// Mitsubishi GX Works2 project: BookEX6_18 Shift   PLC: Q13UDV

// global labels: Global
VAR_GLOBAL
  bVar0 AT M5000 : BOOL;
  abArray0 AT M5010 : ARRAY [0..49] OF BOOL;
  sStr0 AT D5000 : STRING[199];
  sStr1 AT D5100 : STRING[199];
  sStr2 AT D5200 : STRING[199];
  sStr3 AT D5300 : STRING[199];
  sStr4 AT D5400 : STRING[199];
  sStr5 AT D5500 : STRING[199];
  sStr6 AT D5600 : STRING[199];
  sStr7 AT D5700 : STRING[199];
  sStr8 AT D5800 : STRING[199];
  sStr9 AT D5900 : STRING[199];
  iVar0 AT D4500 : INT;
  iVar1 AT D4501 : INT;
  iVar2 AT D4502 : INT;
  iVar3 AT D4503 : INT;
  iVar4 AT D4504 : INT;
  iVar5 AT D4505 : INT;
  iVar6 AT D4506 : INT;
  iVar7 AT D4507 : INT;
  iVar8 AT D4508 : INT;
  iVar9 AT D4509 : INT;
  dVar0 AT D4510 : DINT;
  dVar1 AT D4512 : DINT;
  dVar2 AT D4514 : DINT;
  dVar3 AT D4516 : DINT;
  dVar4 AT D4518 : DINT;
  dVar5 AT D4520 : DINT;
  dVar6 AT D4522 : DINT;
  dVar7 AT D4524 : DINT;
  dVar8 AT D4526 : DINT;
  dVar9 AT D4528 : DINT;
  wVar0 AT D4530 : WORD;
  wVar1 AT D4531 : WORD;
  wVar2 AT D4532 : WORD;
  wVar3 AT D4533 : WORD;
  wVar4 AT D4534 : WORD;
  wVar5 AT D4535 : WORD;
  wVar6 AT D4536 : WORD;
  wVar7 AT D4537 : WORD;
  wVar8 AT D4538 : WORD;
  wVar9 AT D4539 : WORD;
  dwVar0 AT D4540 : DWORD;
  dwVar1 AT D4542 : DWORD;
  dwVar2 AT D4544 : DWORD;
  dwVar3 AT D4546 : DWORD;
  dwVar4 AT D4548 : DWORD;
  dwVar5 AT D4550 : DWORD;
  dwVar6 AT D4552 : DWORD;
  dwVar7 AT D4554 : DWORD;
  dwVar8 AT D4556 : DWORD;
  dwVar9 AT D4558 : DWORD;
  fsVar0 AT D4560 : REAL;
  fsVar1 AT D4562 : REAL;
  fsVar2 AT D4564 : REAL;
  fsVar3 AT D4566 : REAL;
  fsVar4 AT D4568 : REAL;
  fsVar5 AT D4570 : REAL;
  fsVar6 AT D4572 : REAL;
  fsVar7 AT D4574 : REAL;
  fsVar8 AT D4576 : REAL;
  fsVar9 AT D4578 : REAL;
  fdVar0 AT D4580 : LREAL;
  tTime0 AT D4620 : TIME;
  tTime1 AT D4622 : TIME;
  tTime2 AT D4624 : TIME;
  tTime3 AT D4626 : TIME;
  tTime4 AT D4628 : TIME;
  tTime5 AT D4630 : TIME;
  tTime6 AT D4632 : TIME;
  tTime7 AT D4634 : TIME;
  tTime8 AT D4636 : TIME;
  tTime9 AT D4638 : TIME;
  tTime10 AT D4640 : TIME;
  bVar1 AT M5001 : BOOL;
  bVar2 AT M5002 : BOOL;
  bVar3 AT M5003 : BOOL;
  bVar4 AT M5004 : BOOL;
  bVar5 AT M5005 : BOOL;
  bVar6 AT M5006 : BOOL;
  bVar7 AT M5007 : BOOL;
  bVar8 AT M5008 : BOOL;
  bVar9 AT M5009 : BOOL;
  abArray1 AT M5060 : ARRAY [0..49] OF BOOL;
  abArray2 AT M5110 : ARRAY [0..49] OF BOOL;
  abArray3 AT M5160 : ARRAY [0..49] OF BOOL;
  abArray4 AT M5210 : ARRAY [0..49] OF BOOL;
  abArray5 AT M5260 : ARRAY [0..49] OF BOOL;
  abArray6 AT M5310 : ARRAY [0..49] OF BOOL;
  abArray7 AT M5360 : ARRAY [0..49] OF BOOL;
  abArray8 AT M5410 : ARRAY [0..49] OF BOOL;
  abArray9 AT M5460 : ARRAY [0..49] OF BOOL;
  fdVar1 AT D4584 : LREAL;
  fdVar2 AT D4588 : LREAL;
  fdVar3 AT D4592 : LREAL;
  fdVar4 AT D4596 : LREAL;
  fdVar5 AT D4600 : LREAL;
  fdVar6 AT D4604 : LREAL;
  fdVar7 AT D4608 : LREAL;
  fdVar8 AT D4612 : LREAL;
  fdVar9 AT D4616 : LREAL;
  aSendData1 AT D100 : ARRAY [0..9] OF INT;
  aiTxData AT D4000 : ARRAY [0..99] OF INT;
  aiRxData AT D4100 : ARRAY [0..99] OF INT;
  iOpenOK AT D3900 : INT;
  iOpenERR AT D3901 : INT;
  iSendOK AT D3902 : INT;
  iSendERR AT D3903 : INT;
  iCloseOK AT D3906 : INT;
  iCloseERR AT D3907 : INT;
  iRecvOK AT D3904 : INT;
  iRecvERR AT D3905 : INT;
  aiTxData2 AT D4200 : ARRAY [0..99] OF INT;
  aiRxData2 AT D4300 : ARRAY [0..99] OF INT;
  iOpenOK2 AT D3908 : INT;
  iOpenERR2 AT D3909 : INT;
  iSendOK2 AT D3910 : INT;
  iSendERR2 AT D3911 : INT;
  iRecvOK2 AT D3912 : INT;
  iRecvERR2 AT D3913 : INT;
  iCloseOK2 AT D3914 : INT;
  iCloseERR2 AT D3915 : INT;
  iEOpenComp AT D3916 : INT;
  iEOpenReq AT D3917 : INT;
  iERecvFlag AT D3918 : INT;
  iOpenCode AT D3919 : INT;
  iSendCode AT D3920 : INT;
  iRecvCode AT D3921 : INT;
  iCloseCode AT D3922 : INT;
  iOpenCode2 AT D3923 : INT;
  iSendCode2 AT D3924 : INT;
  iRecvCode2 AT D3925 : INT;
  iCloseCode2 AT D3926 : INT;
  aRecvData1 AT D110 : ARRAY [0..9] OF INT;
  aSendData2 AT D120 : ARRAY [0..9] OF INT;
  aRecvData2 AT D130 : ARRAY [0..9] OF INT;
END_VAR
// user libraries (not included): HMI

PROGRAM ExSFT
VAR
  HMI05_1 : HMI05;
END_VAR
(* structured ladder/FBD written out as ST: instructions are called as NAME(EN, inputs, outputs); _pN, _eN, _tN stand for wires *)
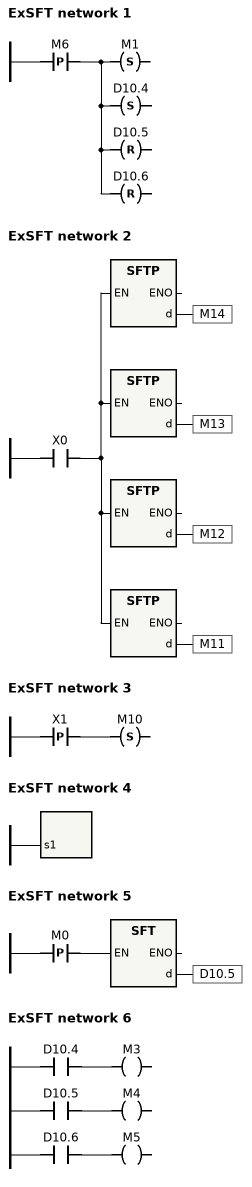
(* network 1 *)
_p1 := LDP(TRUE, M6);
SET(_p1, M1);
SET(_p1, D10.4);
RST(_p1, D10.5);
RST(_p1, D10.6);
(* network 2 *)
SFTP(X0, M14);
SFTP(X0, M13);
SFTP(X0, M12);
SFTP(X0, M11);
(* network 3 *)
SET(LDP(TRUE, X1), M10);
(* network 4 *)
(* element kind 10  <- TRUE *)
(* network 5 *)
SFT(LDP(TRUE, M0), D10.5);
(* network 6 *)
M3 := D10.4;
M4 := D10.5;
M5 := D10.6;
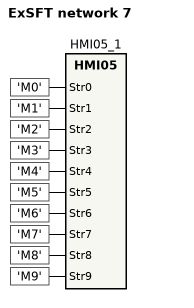
(* network 7 *)
HMI05_1(Str0 := 'M0', Str1 := 'M1', Str2 := 'M2', Str3 := 'M3', Str4 := 'M4', Str5 := 'M5', Str6 := 'M6', Str7 := 'M7', Str8 := 'M8', Str9 := 'M9');
END_PROGRAM

PROGRAM ExWordSFT
VAR
  HMI05_1 : HMI05;
END_VAR
(* structured ladder/FBD written out as ST: instructions are called as NAME(EN, inputs, outputs); _pN, _eN, _tN stand for wires *)
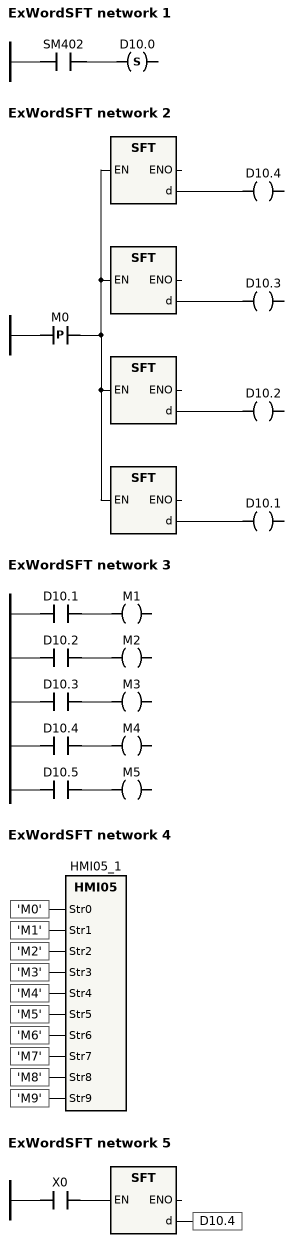
(* network 1 *)
SET(SM402, D10.0);
(* network 2 *)
_p1 := LDP(TRUE, M0);
SFT(_p1, _t2);
D10.4 := _t2;
SFT(_p1, _t3);
D10.3 := _t3;
SFT(_p1, _t4);
D10.2 := _t4;
SFT(_p1, _t5);
D10.1 := _t5;
(* network 3 *)
M1 := D10.1;
M2 := D10.2;
M3 := D10.3;
M4 := D10.4;
M5 := D10.5;
(* network 4 *)
HMI05_1(Str0 := 'M0', Str1 := 'M1', Str2 := 'M2', Str3 := 'M3', Str4 := 'M4', Str5 := 'M5', Str6 := 'M6', Str7 := 'M7', Str8 := 'M8', Str9 := 'M9');
(* network 5 *)
SFT(X0, D10.4);
END_PROGRAM

PROGRAM ExBitSFT
VAR
  HMI05_1 : HMI05;
END_VAR
(* structured ladder/FBD written out as ST: instructions are called as NAME(EN, inputs, outputs); _pN, _eN, _tN stand for wires *)
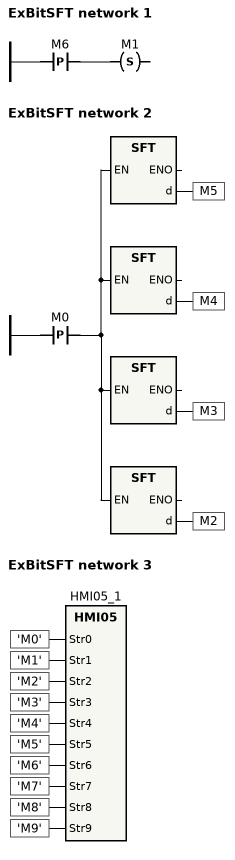
(* network 1 *)
SET(LDP(TRUE, M6), M1);
(* network 2 *)
_p1 := LDP(TRUE, M0);
SFT(_p1, M5);
SFT(_p1, M4);
SFT(_p1, M3);
SFT(_p1, M2);
(* network 3 *)
HMI05_1(Str0 := 'M0', Str1 := 'M1', Str2 := 'M2', Str3 := 'M3', Str4 := 'M4', Str5 := 'M5', Str6 := 'M6', Str7 := 'M7', Str8 := 'M8', Str9 := 'M9');
END_PROGRAM

PROGRAM ExBitSFT2
VAR
  HMI05_1 : HMI05;
END_VAR
(* structured ladder/FBD written out as ST: instructions are called as NAME(EN, inputs, outputs); _pN, _eN, _tN stand for wires *)
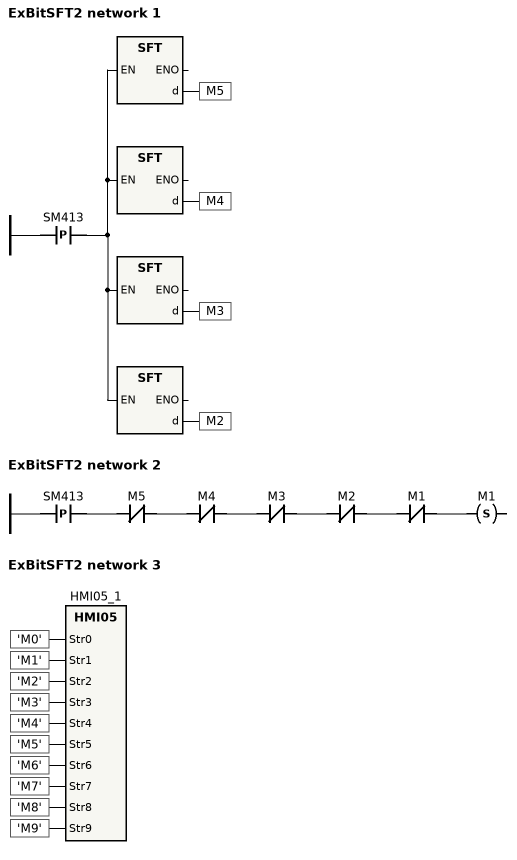
(* network 1 *)
_p1 := LDP(TRUE, SM413);
SFT(_p1, M5);
SFT(_p1, M4);
SFT(_p1, M3);
SFT(_p1, M2);
(* network 2 *)
SET(LDP(TRUE, SM413) AND NOT M5 AND NOT M4 AND NOT M3 AND NOT M2 AND NOT M1, M1);
(* network 3 *)
HMI05_1(Str0 := 'M0', Str1 := 'M1', Str2 := 'M2', Str3 := 'M3', Str4 := 'M4', Str5 := 'M5', Str6 := 'M6', Str7 := 'M7', Str8 := 'M8', Str9 := 'M9');
END_PROGRAM
